// TIA Portal V17 export
// export: Created 2024-08-20T13:26:08.0357762Z, ExportSetting WithDefaults, DisplayName Totally Integrated Automation Portal, DisplayVersion V17 Update 4, DisplayName TIA Portal Openness, DisplayVersion V17 Update 4, DisplayName TIA Portal Version Control Interface, DisplayVersion V17, DisplayName STEP 7 Professional, DisplayVersion V17 Update 4, DisplayName STEP 7 Safety, DisplayVersion V17, DisplayName WinCC Advanced, DisplayVersion V17 Update 4
FUNCTION_BLOCK "LOOP"   // FB2, LAD
{ S7_Optimized_Access := 'TRUE' }
VERSION : 0.1
// stored: AutoNumber true, IsIECCheckEnabled false, IsRetainMemResEnabled false, MemoryReserve 100, SetENOAutomatically false, UDAEnableTagReadback false
   VAR
      PULSO : Bool;
      AuxLoop : Bool;
      N_L00P : Int;
      Aux_N_LOOP : Int;
      Loop : Int;
   END_VAR
   VAR_TEMP   // added for the SCL form of the ladder/FBD networks
      _w1 : Bool;
      _w2 : Bool;
   END_VAR
BEGIN

REGION Network 2
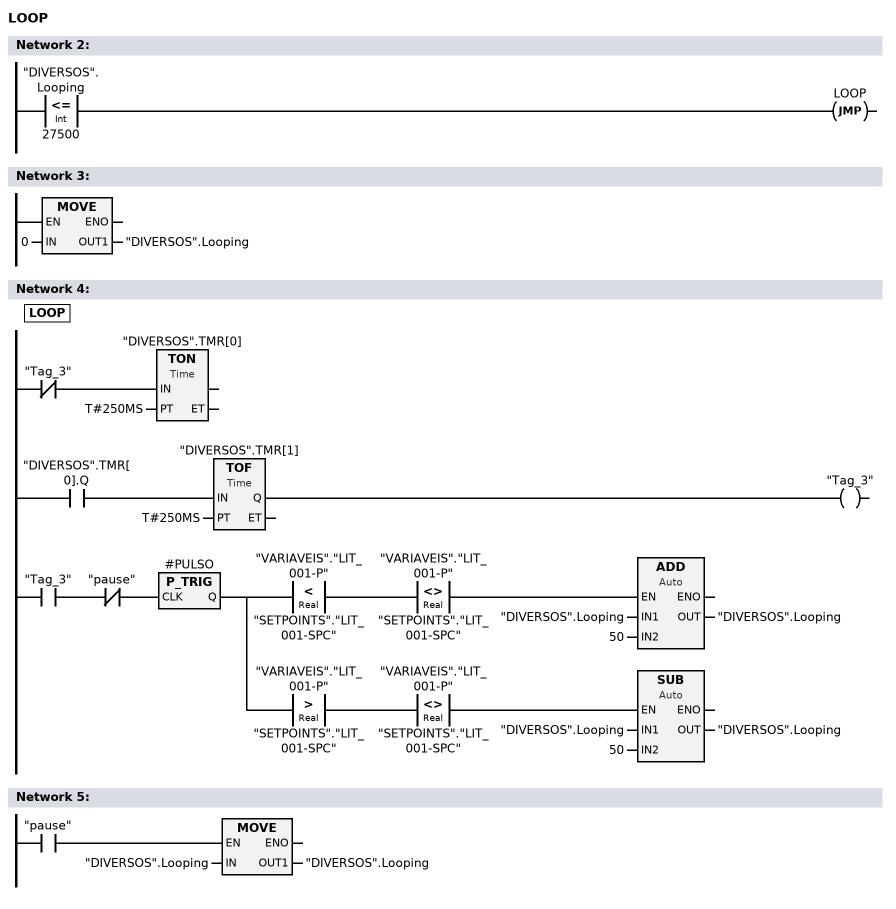
   RUNG wire#powerrail
      { S7_Templates := "SrcType := Int" } LE_Contact(in1 := "DIVERSOS".Looping, in2 := 27500)
      JumpCoil( LOOP )
   END_RUNG
   // the same network as SCL:
   IF "DIVERSOS".Looping <= 27500 THEN GOTO LOOP; END_IF;
END_REGION

REGION Network 3
   RUNG wire#powerrail
      Move(in := 0, out1 => "DIVERSOS".Looping)
   END_RUNG
   // the same network as SCL:
   "DIVERSOS".Looping := 0;
END_REGION

REGION Network 4
   Label( LOOP )
   RUNG wire#powerrail
      I_Contact( "Tag_3" )
      { S7_Templates := "time_type := Time" } "DIVERSOS".TMR[0].TON(pt := T#250MS, et =>)
   END_RUNG
   RUNG wire#powerrail
      Contact( "DIVERSOS".TMR[0].Q )
      { S7_Templates := "time_type := Time" } "DIVERSOS".TMR[1].TOF(pt := T#250MS, et =>)
      Coil( "Tag_3" )
   END_RUNG
   RUNG wire#powerrail
      Contact( "Tag_3" )
      I_Contact( "pause" )
      P_Trig( #PULSO )
      wire#w1
      { S7_Templates := "SrcType := Real" } LT_Contact(in1 := "VARIAVEIS"."LIT_001-P", in2 := "SETPOINTS"."LIT_001-SPC")
      { S7_Templates := "SrcType := Real" } NE_Contact(in1 := "VARIAVEIS"."LIT_001-P", in2 := "SETPOINTS"."LIT_001-SPC")
      Add(in1 := "DIVERSOS".Looping, in2 := 50, out => "DIVERSOS".Looping)
   END_RUNG
   RUNG wire#w1
      { S7_Templates := "SrcType := Real" } GT_Contact(in1 := "VARIAVEIS"."LIT_001-P", in2 := "SETPOINTS"."LIT_001-SPC")
      { S7_Templates := "SrcType := Real" } NE_Contact(in1 := "VARIAVEIS"."LIT_001-P", in2 := "SETPOINTS"."LIT_001-SPC")
      Sub(in1 := "DIVERSOS".Looping, in2 := 50, out => "DIVERSOS".Looping)
   END_RUNG
   // the same network as SCL:
   LOOP:
   "DIVERSOS".TMR[0].TON(IN := NOT "Tag_3", PT := T#250MS);
   "DIVERSOS".TMR[1].TOF(IN := "DIVERSOS".TMR[0].Q, PT := T#250MS);
   "Tag_3" := "DIVERSOS".TMR[1].Q;
   #_w1 := "Tag_3" AND NOT "pause";
   #_w2 := #_w1 AND NOT #PULSO;   // rising edge
   #PULSO := #_w1;
   IF #_w2 AND ("VARIAVEIS"."LIT_001-P" < "SETPOINTS"."LIT_001-SPC") AND ("VARIAVEIS"."LIT_001-P" <> "SETPOINTS"."LIT_001-SPC") THEN
       "DIVERSOS".Looping := "DIVERSOS".Looping + 50;
   END_IF;
   IF #_w2 AND ("VARIAVEIS"."LIT_001-P" > "SETPOINTS"."LIT_001-SPC") AND ("VARIAVEIS"."LIT_001-P" <> "SETPOINTS"."LIT_001-SPC") THEN
       "DIVERSOS".Looping := "DIVERSOS".Looping - 50;
   END_IF;
END_REGION

REGION Network 5
   RUNG wire#powerrail
      Contact( "pause" )
      Move(in := "DIVERSOS".Looping, out1 => "DIVERSOS".Looping)
   END_RUNG
   // the same network as SCL:
   IF "pause" THEN "DIVERSOS".Looping := "DIVERSOS".Looping; END_IF;
END_REGION
END_FUNCTION_BLOCK
